{attribute 'qualified_only'}
{attribute 'strict'}
{attribute 'to_string'}
TYPE TcEventSeverityExt : (
		Verbose	 := 0,
		Info	 := 1,
		Warning	 := 2,
		Error	 := 3,
		Critical := 4,
		Off		 := 5
	);
END_TYPE

(* stored: Version 1.1.0.1
   DUT TcEventSeverityExt: Id {034a2f54-77a8-4290-937a-2f415f361568} *)
